{attribute 'GeneratedUsingTerminal: EK1100-0000-0018'}
{attribute addProperty BoxType "EK1100-0000-0018"}
{attribute addProperty Id "Beckhoff_EL9xxxEK1122Beckhoff_EL9xxxEK1122_0D2A34A32A_0003_EL9110_0000_0016EL9110_2DA353FE5A_0004_EL9110_0000_0017EL9110_2DA353FE5A_0005_EL9110_0000_0018EL9110_2DA353FE5A_0006_EL9160_0000_0016EL9160_2DA353FE5A_0007_EL9210_0000_0016EL9210_B3C0CA836A_0008_EL9210_0000_0017EL9210_B3C0CA836A_0009_EL9210_0000_0018EL9210_B3C0CA836A_0010_EL9210_0020_0016EL9210_B3C0CA836A_0011_EL9210_0020_0017EL9210_B3C0CA836A_0012_EL9210_0020_0018EL9210_B3C0CA836A_0013_EL9221_4030_0018EL9221_8223B8D725A_0014_EL9221_5000_0018EL9221_8223B8D725A_0015_EL9221_5090_0018EL9221_8223B8D725A_0016_EL9221_6000_0018EL9221_8223B8D725A_0017_EL9221_6040_0018EL9221_8223B8D725A_0018_EL9221_9060_0018EL9221_8223B8D725A_0019_EL9221_9080_0018EL9221_8223B8D725A_0020_EL9222_4433_0018EL9222_621C429E38A_0021_EL9222_5500_0018EL9222_621C429E38A_0022_EL9222_6600_0018EL9222_621C429E38A_0023_EL9222_6644_0018EL9222_621C429E38A_0024_EL9222_9482_0018EL9222_621C429E38A_0025_EL9222_9664_0018EL9222_621C429E38A_0026_EL9227_4433_0018EL9227_5EE3BA1D72A_0027_EL9227_5500_0018EL9227_5EE3BA1D72A_0028_EL9227_6600_0018EL9227_5EE3BA1D72A_0029_EL9227_6644_0018EL9227_5EE3BA1D72A_0030_EL9227_9482_0018EL9227_5EE3BA1D72A_0031_EL9227_9664_0018EL9227_5EE3BA1D72A_0032_EL9260_0000_0016EL9260_B3C0CA836A_0033_EL9410_0000_0016EL9410_6BC01D146A_0034_EL9410_0000_0017EL9410_6BC01D146A_0035_EL9505_0000_0016EL9505_19A4723D6A_0036_EL9505_0000_0017EL9505_19A4723D6A_0037_EL9505_0000_0018EL9505_19A4723D6A_0038_EL9508_0000_0016EL9508_19A4723D6A_0039_EL9508_0000_0017EL9508_19A4723D6A_0040_EL9508_0000_0018EL9508_19A4723D6A_0041_EL9510_0000_0016EL9510_19A4723D6A_0042_EL9510_0000_0017EL9510_19A4723D6A_0043_EL9510_0000_0018EL9510_19A4723D6A_0044_EL9512_0000_0016EL9512_19A4723D6A_0045_EL9512_0000_0017EL9512_19A4723D6A_0046_EL9512_0000_0018EL9512_19A4723D6A_0047_EL9515_0000_0016EL9515_19A4723D6A_0048_EL9515_0000_0017EL9515_19A4723D6A_0049_EL9515_0000_0018EL9515_19A4723D6A_0050_EL9520_0000_0016EL9520_C0C35FE85A_0051_EL9520_0000_0017EL9520_C0C35FE85A_0052_EL9540_0010_0016EL9540_67D07E0A6A_0053_EL9550_0010_0016EL9550_3E8321A98A_0054_EL9560_0000_0016EL9560_DD45A30A6A_0055_EL9560_0000_0017EL9560_DD45A30A6A_0056_EL9560_0000_0018EL9560_DD45A30A6A_0057_EL9576_0000_0016EL9576_1C51438027A_0058_EL9576_0000_0017EL9576_6D7359CA28A_0059_EL9576_0000_0018EL9576_6D7359CA28A_0060_EL9576_0000_0019EL9576_85AB580429A_0061_EL9576_0000_0020EL9576_1017F4A528A_0062_EL9576_0000_0021EL9576_1017F4A528A_0063_EL9576_0000_0022EL9576_C42142C629A_0086_EL9540_0010EL9540_67D07E0A6A_0088_EL9550_0010EL9550_3E8321A98"}
{attribute addProperty CRC "2540816684"}
{attribute addProperty Size "1254"}
TYPE Beckhoff_EL9xxx_9771C92C EXTENDS EK1100_1FC0878B :
STRUCT
	{attribute addProperty Name "Beckhoff EL9xxxEK1122"}
	{attribute addProperty PreviousPort "Beckhoff EL9xxx : B"}
	Beckhoff_EL9xxxEK1122 : Beckhoff_EL9xxxEK1122_0D2A34A3;
	{attribute addProperty Name "A_0003(EL9110-0000-0016)"}
	{attribute addProperty PreviousPort "Beckhoff EL9xxxEK1122 : C"}
	A_0003_EL9110_0000_0016 : EL9110_2DA353FE;
	{attribute addProperty Name "A_0004(EL9110-0000-0017)"}
	{attribute addProperty PreviousPort "A_0003(EL9110-0000-0016) : B"}
	A_0004_EL9110_0000_0017 : EL9110_2DA353FE;
	{attribute addProperty Name "A_0005(EL9110-0000-0018)"}
	{attribute addProperty PreviousPort "A_0004(EL9110-0000-0017) : B"}
	A_0005_EL9110_0000_0018 : EL9110_2DA353FE;
	{attribute addProperty Name "A_0006(EL9160-0000-0016)"}
	{attribute addProperty PreviousPort "A_0005(EL9110-0000-0018) : B"}
	A_0006_EL9160_0000_0016 : EL9160_2DA353FE;
	{attribute addProperty Name "A_0007(EL9210-0000-0016)"}
	{attribute addProperty PreviousPort "A_0006(EL9160-0000-0016) : B"}
	A_0007_EL9210_0000_0016 : EL9210_B3C0CA83;
	{attribute addProperty Name "A_0008(EL9210-0000-0017)"}
	{attribute addProperty PreviousPort "A_0007(EL9210-0000-0016) : B"}
	A_0008_EL9210_0000_0017 : EL9210_B3C0CA83;
	{attribute addProperty Name "A_0009(EL9210-0000-0018)"}
	{attribute addProperty PreviousPort "A_0008(EL9210-0000-0017) : B"}
	A_0009_EL9210_0000_0018 : EL9210_B3C0CA83;
	{attribute addProperty Name "A_0010(EL9210-0020-0016)"}
	{attribute addProperty PreviousPort "A_0009(EL9210-0000-0018) : B"}
	A_0010_EL9210_0020_0016 : EL9210_B3C0CA83;
	{attribute addProperty Name "A_0011(EL9210-0020-0017)"}
	{attribute addProperty PreviousPort "A_0010(EL9210-0020-0016) : B"}
	A_0011_EL9210_0020_0017 : EL9210_B3C0CA83;
	{attribute addProperty Name "A_0012(EL9210-0020-0018)"}
	{attribute addProperty PreviousPort "A_0011(EL9210-0020-0017) : B"}
	A_0012_EL9210_0020_0018 : EL9210_B3C0CA83;
	{attribute addProperty Name "A_0013(EL9221-4030-0018)"}
	{attribute addProperty PreviousPort "A_0012(EL9210-0020-0018) : B"}
	A_0013_EL9221_4030_0018 : EL9221_8223B8D7;
	{attribute addProperty Name "A_0014(EL9221-5000-0018)"}
	{attribute addProperty PreviousPort "A_0013(EL9221-4030-0018) : B"}
	A_0014_EL9221_5000_0018 : EL9221_8223B8D7;
	{attribute addProperty Name "A_0015(EL9221-5090-0018)"}
	{attribute addProperty PreviousPort "A_0014(EL9221-5000-0018) : B"}
	A_0015_EL9221_5090_0018 : EL9221_8223B8D7;
	{attribute addProperty Name "A_0016(EL9221-6000-0018)"}
	{attribute addProperty PreviousPort "A_0015(EL9221-5090-0018) : B"}
	A_0016_EL9221_6000_0018 : EL9221_8223B8D7;
	{attribute addProperty Name "A_0017(EL9221-6040-0018)"}
	{attribute addProperty PreviousPort "A_0016(EL9221-6000-0018) : B"}
	A_0017_EL9221_6040_0018 : EL9221_8223B8D7;
	{attribute addProperty Name "A_0018(EL9221-9060-0018)"}
	{attribute addProperty PreviousPort "A_0017(EL9221-6040-0018) : B"}
	A_0018_EL9221_9060_0018 : EL9221_8223B8D7;
	{attribute addProperty Name "A_0019(EL9221-9080-0018)"}
	{attribute addProperty PreviousPort "A_0018(EL9221-9060-0018) : B"}
	A_0019_EL9221_9080_0018 : EL9221_8223B8D7;
	{attribute addProperty Name "A_0020(EL9222-4433-0018)"}
	{attribute addProperty PreviousPort "A_0019(EL9221-9080-0018) : B"}
	A_0020_EL9222_4433_0018 : EL9222_621C429E;
	{attribute addProperty Name "A_0021(EL9222-5500-0018)"}
	{attribute addProperty PreviousPort "A_0020(EL9222-4433-0018) : B"}
	A_0021_EL9222_5500_0018 : EL9222_621C429E;
	{attribute addProperty Name "A_0022(EL9222-6600-0018)"}
	{attribute addProperty PreviousPort "A_0021(EL9222-5500-0018) : B"}
	A_0022_EL9222_6600_0018 : EL9222_621C429E;
	{attribute addProperty Name "A_0023(EL9222-6644-0018)"}
	{attribute addProperty PreviousPort "A_0022(EL9222-6600-0018) : B"}
	A_0023_EL9222_6644_0018 : EL9222_621C429E;
	{attribute addProperty Name "A_0024(EL9222-9482-0018)"}
	{attribute addProperty PreviousPort "A_0023(EL9222-6644-0018) : B"}
	A_0024_EL9222_9482_0018 : EL9222_621C429E;
	{attribute addProperty Name "A_0025(EL9222-9664-0018)"}
	{attribute addProperty PreviousPort "A_0024(EL9222-9482-0018) : B"}
	A_0025_EL9222_9664_0018 : EL9222_621C429E;
	{attribute addProperty Name "A_0026(EL9227-4433-0018)"}
	{attribute addProperty PreviousPort "A_0025(EL9222-9664-0018) : B"}
	A_0026_EL9227_4433_0018 : EL9227_5EE3BA1D;
	{attribute addProperty Name "A_0027(EL9227-5500-0018)"}
	{attribute addProperty PreviousPort "A_0026(EL9227-4433-0018) : B"}
	A_0027_EL9227_5500_0018 : EL9227_5EE3BA1D;
	{attribute addProperty Name "A_0028(EL9227-6600-0018)"}
	{attribute addProperty PreviousPort "A_0027(EL9227-5500-0018) : B"}
	A_0028_EL9227_6600_0018 : EL9227_5EE3BA1D;
	{attribute addProperty Name "A_0029(EL9227-6644-0018)"}
	{attribute addProperty PreviousPort "A_0028(EL9227-6600-0018) : B"}
	A_0029_EL9227_6644_0018 : EL9227_5EE3BA1D;
	{attribute addProperty Name "A_0030(EL9227-9482-0018)"}
	{attribute addProperty PreviousPort "A_0029(EL9227-6644-0018) : B"}
	A_0030_EL9227_9482_0018 : EL9227_5EE3BA1D;
	{attribute addProperty Name "A_0031(EL9227-9664-0018)"}
	{attribute addProperty PreviousPort "A_0030(EL9227-9482-0018) : B"}
	A_0031_EL9227_9664_0018 : EL9227_5EE3BA1D;
	{attribute addProperty Name "A_0032(EL9260-0000-0016)"}
	{attribute addProperty PreviousPort "A_0031(EL9227-9664-0018) : B"}
	A_0032_EL9260_0000_0016 : EL9260_B3C0CA83;
	{attribute addProperty Name "A_0033(EL9410-0000-0016)"}
	{attribute addProperty PreviousPort "A_0032(EL9260-0000-0016) : B"}
	A_0033_EL9410_0000_0016 : EL9410_6BC01D14;
	{attribute addProperty Name "A_0034(EL9410-0000-0017)"}
	{attribute addProperty PreviousPort "A_0033(EL9410-0000-0016) : B"}
	A_0034_EL9410_0000_0017 : EL9410_6BC01D14;
	{attribute addProperty Name "A_0035(EL9505-0000-0016)"}
	{attribute addProperty PreviousPort "A_0034(EL9410-0000-0017) : B"}
	A_0035_EL9505_0000_0016 : EL9505_19A4723D;
	{attribute addProperty Name "A_0036(EL9505-0000-0017)"}
	{attribute addProperty PreviousPort "A_0035(EL9505-0000-0016) : B"}
	A_0036_EL9505_0000_0017 : EL9505_19A4723D;
	{attribute addProperty Name "A_0037(EL9505-0000-0018)"}
	{attribute addProperty PreviousPort "A_0036(EL9505-0000-0017) : B"}
	A_0037_EL9505_0000_0018 : EL9505_19A4723D;
	{attribute addProperty Name "A_0038(EL9508-0000-0016)"}
	{attribute addProperty PreviousPort "A_0037(EL9505-0000-0018) : B"}
	A_0038_EL9508_0000_0016 : EL9508_19A4723D;
	{attribute addProperty Name "A_0039(EL9508-0000-0017)"}
	{attribute addProperty PreviousPort "A_0038(EL9508-0000-0016) : B"}
	A_0039_EL9508_0000_0017 : EL9508_19A4723D;
	{attribute addProperty Name "A_0040(EL9508-0000-0018)"}
	{attribute addProperty PreviousPort "A_0039(EL9508-0000-0017) : B"}
	A_0040_EL9508_0000_0018 : EL9508_19A4723D;
	{attribute addProperty Name "A_0041(EL9510-0000-0016)"}
	{attribute addProperty PreviousPort "A_0040(EL9508-0000-0018) : B"}
	A_0041_EL9510_0000_0016 : EL9510_19A4723D;
	{attribute addProperty Name "A_0042(EL9510-0000-0017)"}
	{attribute addProperty PreviousPort "A_0041(EL9510-0000-0016) : B"}
	A_0042_EL9510_0000_0017 : EL9510_19A4723D;
	{attribute addProperty Name "A_0043(EL9510-0000-0018)"}
	{attribute addProperty PreviousPort "A_0042(EL9510-0000-0017) : B"}
	A_0043_EL9510_0000_0018 : EL9510_19A4723D;
	{attribute addProperty Name "A_0044(EL9512-0000-0016)"}
	{attribute addProperty PreviousPort "A_0043(EL9510-0000-0018) : B"}
	A_0044_EL9512_0000_0016 : EL9512_19A4723D;
	{attribute addProperty Name "A_0045(EL9512-0000-0017)"}
	{attribute addProperty PreviousPort "A_0044(EL9512-0000-0016) : B"}
	A_0045_EL9512_0000_0017 : EL9512_19A4723D;
	{attribute addProperty Name "A_0046(EL9512-0000-0018)"}
	{attribute addProperty PreviousPort "A_0045(EL9512-0000-0017) : B"}
	A_0046_EL9512_0000_0018 : EL9512_19A4723D;
	{attribute addProperty Name "A_0047(EL9515-0000-0016)"}
	{attribute addProperty PreviousPort "A_0046(EL9512-0000-0018) : B"}
	A_0047_EL9515_0000_0016 : EL9515_19A4723D;
	{attribute addProperty Name "A_0048(EL9515-0000-0017)"}
	{attribute addProperty PreviousPort "A_0047(EL9515-0000-0016) : B"}
	A_0048_EL9515_0000_0017 : EL9515_19A4723D;
	{attribute addProperty Name "A_0049(EL9515-0000-0018)"}
	{attribute addProperty PreviousPort "A_0048(EL9515-0000-0017) : B"}
	A_0049_EL9515_0000_0018 : EL9515_19A4723D;
	{attribute addProperty Name "A_0050(EL9520-0000-0016)"}
	{attribute addProperty PreviousPort "A_0049(EL9515-0000-0018) : B"}
	A_0050_EL9520_0000_0016 : EL9520_C0C35FE8;
	{attribute addProperty Name "A_0051(EL9520-0000-0017)"}
	{attribute addProperty PreviousPort "A_0050(EL9520-0000-0016) : B"}
	A_0051_EL9520_0000_0017 : EL9520_C0C35FE8;
	{attribute addProperty Name "A_0052(EL9540-0010-0016)"}
	{attribute addProperty PreviousPort "A_0051(EL9520-0000-0017) : B"}
	A_0052_EL9540_0010_0016 : EL9540_67D07E0A;
	{attribute addProperty Name "A_0053(EL9550-0010-0016)"}
	{attribute addProperty PreviousPort "A_0052(EL9540-0010-0016) : B"}
	A_0053_EL9550_0010_0016 : EL9550_3E8321A9;
	{attribute addProperty Name "A_0054(EL9560-0000-0016)"}
	{attribute addProperty PreviousPort "A_0053(EL9550-0010-0016) : B"}
	A_0054_EL9560_0000_0016 : EL9560_DD45A30A;
	{attribute addProperty Name "A_0055(EL9560-0000-0017)"}
	{attribute addProperty PreviousPort "A_0054(EL9560-0000-0016) : B"}
	A_0055_EL9560_0000_0017 : EL9560_DD45A30A;
	{attribute addProperty Name "A_0056(EL9560-0000-0018)"}
	{attribute addProperty PreviousPort "A_0055(EL9560-0000-0017) : B"}
	A_0056_EL9560_0000_0018 : EL9560_DD45A30A;
	{attribute addProperty Name "A_0057(EL9576-0000-0016)"}
	{attribute addProperty PreviousPort "A_0056(EL9560-0000-0018) : B"}
	A_0057_EL9576_0000_0016 : EL9576_1C514380;
	{attribute addProperty Name "A_0058(EL9576-0000-0017)"}
	{attribute addProperty PreviousPort "A_0057(EL9576-0000-0016) : B"}
	A_0058_EL9576_0000_0017 : EL9576_6D7359CA;
	{attribute addProperty Name "A_0059(EL9576-0000-0018)"}
	{attribute addProperty PreviousPort "A_0058(EL9576-0000-0017) : B"}
	A_0059_EL9576_0000_0018 : EL9576_6D7359CA;
	{attribute addProperty Name "A_0060(EL9576-0000-0019)"}
	{attribute addProperty PreviousPort "A_0059(EL9576-0000-0018) : B"}
	A_0060_EL9576_0000_0019 : EL9576_85AB5804;
	{attribute addProperty Name "A_0061(EL9576-0000-0020)"}
	{attribute addProperty PreviousPort "A_0060(EL9576-0000-0019) : B"}
	A_0061_EL9576_0000_0020 : EL9576_1017F4A5;
	{attribute addProperty Name "A_0062(EL9576-0000-0021)"}
	{attribute addProperty PreviousPort "A_0061(EL9576-0000-0020) : B"}
	A_0062_EL9576_0000_0021 : EL9576_1017F4A5;
	{attribute addProperty Name "A_0063(EL9576-0000-0022)"}
	{attribute addProperty PreviousPort "A_0062(EL9576-0000-0021) : B"}
	A_0063_EL9576_0000_0022 : EL9576_C42142C6;
	{attribute addProperty Name "A_0086 (EL9540-0010)"}
	{attribute addProperty PreviousPort "A_0063(EL9576-0000-0022) : B"}
	A_0086_EL9540_0010 : EL9540_67D07E0A;
	{attribute addProperty Name "A_0088 (EL9550-0010)"}
	{attribute addProperty PreviousPort "A_0086 (EL9540-0010) : B"}
	A_0088_EL9550_0010 : EL9550_3E8321A9;
END_STRUCT
END_TYPE

(* stored: Version 1.2.0.0, ProductVersion 3.1.4024.9
   DUT Beckhoff_EL9xxx_9771C92C: Id {d75b8ed5-cc1d-4da4-9697-a83d39a3d473} *)
